(* IEC 61131-3 sources: repolevel_ST_code_completion/real_groud_truth最新/repoeval_Interation_HowTo/full_result, 2 files *)

(* ---- FirstPublish.st ---- *)
FUNCTION_BLOCK FirstPublish
VAR_INPUT
END_VAR
VAR_OUTPUT
END_VAR

VAR
    publisher: MQTT.MQTTPublish;
    init: BOOL;
END_VAR

IF NOT init THEN
    init := TRUE;
    publisher.SetMqttInOut(MQTT_IN_OUT := HowTo.MQTT_IN_OUT);
END_IF

publisher(
    Publish := TRUE,
    Topic := ADR('TestTopic/FromCodesys'),
    Payload := ADR('Hello from Codesys!'),
    QoSPublish := MQTT.QoS.ExactlyOnce,
    Retain := FALSE);
END_FUNCTION_BLOCK

(* ---- FirstSubscription.st ---- *)
FUNCTION_BLOCK FirstSubscription
VAR_INPUT
END_VAR
VAR_OUTPUT
END_VAR

VAR
    subscriber: MQTT.MQTTSubscribe;
    init: BOOL;
    receivedPayload: STRING;
    doSubscribe: BOOL;
END_VAR

IF NOT init THEN
    init := TRUE;
    subscriber.SetMqttInOut(MQTT_IN_OUT := HowTo.MQTT_IN_OUT);
END_IF

subscriber(
    Topic := ADR('TestTopic/FromCodesys'),
    PayloadString := ADR(receivedPayload),
    SubscribeAsString := TRUE,
    QoSIn := MQTT.QoS.ExactlyOnce,
    send := doSubscribe);
END_FUNCTION_BLOCK
